FUNCTION_BLOCK FB_testAxle 
VAR
 	stm	: UINT := 10;
  stmAfterInit : UINT := 1000;
  stIRL : ST_LineReference;
  bFW, bBW : BOOL := FALSE;
END_VAR

G.AxisLine1Front(); 
G.AxisLine2Front();
G.AxisLine1Back();
G.AxisLine2Back();
G.AxisMaster();

CASE stm OF   
  10:
    stIRL.nThis := 0;
    stIRL.nFixedID := 1;
    G.AxisLine1Front.Init(stIrrLine := stIRL, stAxisMotor_R := ADR(G.stAX.Line1Front), stAxisMaster_R := ADR(G.stAX.Master));
    G.AxisLine2Front.Init(stIrrLine := stIRL, stAxisMotor_R := ADR(G.stAX.Line2Front), stAxisMaster_R := ADR(G.stAX.Master));
    G.AxisLine1Back.Init(stIrrLine := stIRL, stAxisMotor_R := ADR(G.stAX.Line1Back), stAxisMaster_R := ADR(G.stAX.Master));
    G.AxisLine2Back.Init(stIrrLine := stIRL, stAxisMotor_R := ADR(G.stAX.Line2Back), stAxisMaster_R := ADR(G.stAX.Master));
    G.AxisMaster.Init(stIrrLine := stIRL, stAxisMotor_R := ADR(G.stAX.Master), stAxisMaster_R := ADR(G.stAX.Master));
   stm := stmAfterInit;

  50:
    IF NOT G.AxisMaster.IsBusy THEN
      G.AxisMaster.RequPowerOn();
      stm := 60;
    END_IF
  60:
    IF G.AxisMaster.IsDone THEN
      stm := 70;
    END_IF
  70:
    IF NOT G.AxisMaster.IsError THEN
      stm := 100;
    ELSE
      stm := 0;
    END_IF

  100:
    IF NOT G.AxisLine1Front.IsBusy THEN
      G.AxisLine1Front.RequPowerOn();
      stm := 120;
    END_IF
  120:
    IF G.AxisLine1Front.IsDone THEN
      stm := 130;
    END_IF
  130:
    IF NOT G.AxisLine1Front.IsError THEN
      stm := 140;
      stm := 0;
    ELSE
      stm := 0;
    END_IF
 
  1000:
    IF NOT G.AxisLine1Front.IsBusy AND NOT G.AxisLine2Front.IsBusy AND NOT G.AxisLine1Back.IsBusy AND NOT G.AxisLine2Back.IsBusy AND NOT G.AxisMaster.IsBusy THEN
      G.AxisLine1Front.RequPowerOn();
      G.AxisLine2Front.RequPowerOn();
      G.AxisLine1Back.RequPowerOn();
      G.AxisLine2Back.RequPowerOn();
      G.AxisMaster.RequPowerOn();
      stm := 1120;
    END_IF
  1120:
    IF G.AxisLine1Front.IsDone AND G.AxisLine2Front.IsDone AND G.AxisLine1Back.IsDone AND G.AxisLine2Back.IsDone AND G.AxisMaster.IsDone THEN
      stm := 1130;
    END_IF
  1130:
    IF NOT G.AxisLine1Front.IsError AND NOT G.AxisLine2Front.IsError AND NOT G.AxisLine1Back.IsError AND NOT G.AxisLine2Back.IsError AND NOT G.AxisMaster.IsError THEN
      stm := 1140;
      stm := 0;
    ELSE
      stm := 0;
    END_IF

  
  140:
    IF NOT G.AxisLine1Front.IsBusy THEN
      G.AxisLine1Front.RequGearInDyn();
      stm := 150;
    END_IF
  150:
    IF G.AxisLine1Front.IsDone THEN
      stm := 160;
    END_IF
  160:
    IF NOT G.AxisLine1Front.IsError THEN
      stm := 170; 
    ELSE
      stm := 0;
    END_IF
    
  170:
    IF NOT G.AxisMaster.IsBusy THEN
      G.AxisMaster.RequJogAxisMaster();
      stm := 180;
    END_IF
  
  180:
    bFW := FALSE;
    bBW := FALSE;
    G.AxisMaster.JogExec(bExecIn := TRUE, bExecJogFWIn := bFW, bExecJogBWIn := bBW);
    stm := 180;
  
  0:; //park 
END_CASE

END_FUNCTION_BLOCK

(* stored: Version 1.1.0.1, ProductVersion 3.1.4024.12
   POU FB_testAxle: Id {9bd3fa27-2c86-4015-af85-c6190e6bedf9}, SpecialFunc None *)
